{attribute 'GeneratedUsingTerminal: EK1122-0000-0018'}
{attribute addProperty BoxType "EK1122-0000-0018"}
{attribute addProperty Id "Beckhoff_EL5xxxsub_EK1100EK1100_AB5A94672"}
{attribute addProperty CRC "2201125532"}
{attribute addProperty Size "2"}
TYPE Beckhoff_EL5xxxEK1122_8332829C EXTENDS EK1122_AB5A9467 :
STRUCT
	{attribute addProperty Name "Beckhoff_EL5xxxsub_EK1100"}
	{attribute addProperty PreviousPort "Beckhoff EL5xxxEK1122 : D"}
	Beckhoff_EL5xxxsub_EK1100 : EK1100_AB5A9467;
END_STRUCT
END_TYPE

(* stored: Version 1.2.0.0, ProductVersion 3.1.4024.9
   DUT Beckhoff_EL5xxxEK1122_8332829C: Id {223dba76-3bd7-4d42-8d53-75ef2fd462dc} *)
